FUNCTION_BLOCK FB_PackMLBase
VAR_INPUT
	PackMLIn	: ST_PML_Base_In;
	
	bEnable				: BOOL := TRUE;
	bExternalFault		: BOOL;
END_VAR
VAR_OUTPUT
	PackMLOut	: ST_PML_Base_Out;
	
	bTransitionActive	: BOOL;
END_VAR
VAR
	_eLastCommand			: E_PackMLCommand := E_PackMLCommand.None;
	_eCommandToProcess		: E_PackMLCommand := E_PackMLCommand.None;
	_eQueuedCommand			: E_PackMLCommand := E_PackMLCommand.None;
	_bQueuedCommandRequest	: BOOL;
	_bCommandConsumed		: BOOL;
	_bModeChangeConsumed	: BOOL;
	_bStateFirstScan		: BOOL := TRUE;
	_bStateFirstScanForHook	: BOOL;
	_eHookResult			: E_PackMLHookResult;
END_VAR

// Reset edge-style status before evaluating this PLC cycle.
_eCommandToProcess		:= E_PackMLCommand.None;

// Command and mode request feedback is latched for HMI/upper-layer handshakes
// until the corresponding request input returns to FALSE.
IF NOT PackMLIn.bCommandChangeRequest THEN
	PackMLOut.bCommandAccepted	:= FALSE;
	PackMLOut.bCommandRejected	:= FALSE;
	PackMLOut.eStateErrorID			:= E_PackMLErrorID.NoError;
END_IF

IF NOT PackMLIn.bModeChangeRequest THEN
	PackMLOut.bModeChanged		:= FALSE;
	PackMLOut.bModeChangeRejected	:= FALSE;
	PackMLOut.eModeErrorID		:= E_PackMLErrorID.NoError;
END_IF

// A disabled base FB holds the current state and suppresses transition activity.
IF NOT bEnable THEN
	bTransitionActive := FALSE;
	RETURN;
END_IF

// Mode change requests are edge/latch based, matching command request behavior.
// The caller must clear stIn.bModeChangeRequest before the same request can run again.
IF NOT PackMLIn.bModeChangeRequest THEN
	_bModeChangeConsumed := FALSE;
END_IF

IF PackMLIn.bModeChangeRequest AND NOT _bModeChangeConsumed THEN
	_bModeChangeConsumed := TRUE;

	IF NOT H_IsModeSupported(PackMLIn.eMode) THEN
		M_RejectModeChange(E_PackMLErrorID.ModeNotSupported);
	ELSIF PackMLIn.eMode = PackMLOut.eModeCurrent THEN
		M_RejectModeChange(E_PackMLErrorID.ModeAlreadyActive);
	ELSIF NOT M_IsModeChangeAllowedByState() THEN
		M_RejectModeChange(E_PackMLErrorID.ModeChangeNotAllowedFromCurrentState);
	ELSIF NOT H_IsStateSupportedByMode(PackMLIn.eMode, PackMLOut.eStateCurrent) THEN
		M_RejectModeChange(E_PackMLErrorID.ModeDoesNotSupportCurrentState);
	ELSE
		M_ChangeMode(PackMLIn.eMode);
	END_IF
END_IF

// Command requests are edge/latch based, matching mode-change request behavior.
// The caller must clear stIn.bCommandChangeRequest before another command can run.
IF NOT PackMLIn.bCommandChangeRequest THEN
	_bCommandConsumed	:= FALSE;
	_eLastCommand		:= E_PackMLCommand.None;
END_IF

// External faults have priority over normal commands and force the abort path
// only while the machine is not already Aborting or Aborted.
IF bExternalFault AND M_IsAbortAllowedByState() THEN
	_eCommandToProcess := E_PackMLCommand.Abort;
ELSIF _bQueuedCommandRequest AND (_eQueuedCommand <> E_PackMLCommand.None) THEN
	_eCommandToProcess		:= _eQueuedCommand;
	_eQueuedCommand			:= E_PackMLCommand.None;
	_bQueuedCommandRequest	:= FALSE;
ELSIF PackMLIn.bCommandChangeRequest AND (PackMLIn.eCommand <> E_PackMLCommand.None) AND NOT _bCommandConsumed THEN
	_eCommandToProcess	:= PackMLIn.eCommand;
	_eLastCommand		:= PackMLIn.eCommand;
	_bCommandConsumed	:= TRUE;
END_IF

// Mode policy hooks run before PackML state guards so a forbidden command reports
// the mode reason instead of a state reason.
IF (_eCommandToProcess <> E_PackMLCommand.None) AND NOT H_IsCommandAllowedByMode(_eCommandToProcess, PackMLOut.eModeCurrent) THEN
	M_RejectCommand(E_PackMLErrorID.CommandNotAllowedInActiveMode);
	_eCommandToProcess := E_PackMLCommand.None;
END_IF

// Dispatch the accepted command through private PackML state guards.
// Rejected commands never mutate the state and return a stable numeric error ID.
CASE _eCommandToProcess OF
	E_PackMLCommand.Clear:
		IF M_IsClearAllowedByState() THEN
			PackMLOut.bCommandAccepted := TRUE;
			M_ChangeState(E_PackMLState.Clearing);
		ELSE
			M_RejectCommand(E_PackMLErrorID.ClearNotAllowedFromCurrentState);
		END_IF

	E_PackMLCommand.Reset:
		IF M_IsResetAllowedByState() THEN
			PackMLOut.bCommandAccepted := TRUE;
			M_ChangeState(E_PackMLState.Resetting);
		ELSE
			M_RejectCommand(E_PackMLErrorID.ResetNotAllowedFromCurrentState);
		END_IF

	E_PackMLCommand.Start:
		IF M_IsStartAllowedByState() THEN
			PackMLOut.bCommandAccepted := TRUE;
			M_ChangeState(E_PackMLState.Starting);
		ELSE
			M_RejectCommand(E_PackMLErrorID.StartNotAllowedFromCurrentState);
		END_IF

	E_PackMLCommand.Stop:
		IF M_IsStopAllowedByState() THEN
			PackMLOut.bCommandAccepted := TRUE;
			M_ChangeState(E_PackMLState.Stopping);
		ELSE
			M_RejectCommand(E_PackMLErrorID.StopNotAllowedFromCurrentState);
		END_IF

	E_PackMLCommand.Hold:
		IF M_IsHoldAllowedByState() THEN
			PackMLOut.bCommandAccepted := TRUE;
			M_ChangeState(E_PackMLState.Holding);
		ELSE
			M_RejectCommand(E_PackMLErrorID.HoldNotAllowedFromCurrentState);
		END_IF

	E_PackMLCommand.Unhold:
		IF M_IsUnholdAllowedByState() THEN
			PackMLOut.bCommandAccepted := TRUE;
			M_ChangeState(E_PackMLState.Unholding);
		ELSE
			M_RejectCommand(E_PackMLErrorID.UnholdNotAllowedFromCurrentState);
		END_IF

	E_PackMLCommand.Suspend:
		IF M_IsSuspendAllowedByState() THEN
			PackMLOut.bCommandAccepted := TRUE;
			M_ChangeState(E_PackMLState.Suspending);
		ELSE
			M_RejectCommand(E_PackMLErrorID.SuspendNotAllowedFromCurrentState);
		END_IF

	E_PackMLCommand.Unsuspend:
		IF M_IsUnsuspendAllowedByState() THEN
			PackMLOut.bCommandAccepted := TRUE;
			M_ChangeState(E_PackMLState.Unsuspending);
		ELSE
			M_RejectCommand(E_PackMLErrorID.UnsuspendNotAllowedFromCurrentState);
		END_IF

	E_PackMLCommand.Abort:
		IF M_IsAbortAllowedByState() THEN
			PackMLOut.bCommandAccepted := TRUE;
			M_ChangeState(E_PackMLState.Aborting);
		ELSE
			M_RejectCommand(E_PackMLErrorID.AbortNotAllowedFromCurrentState);
		END_IF
END_CASE

// Run the current state's action hook, then advance transient states when their
// hook reports Done. Stable states remain active until a command moves them.
_bStateFirstScanForHook	:= _bStateFirstScan;
_bStateFirstScan		:= FALSE;

CASE PackMLOut.eStateCurrent OF
	E_PackMLState.Undefined:
		_eHookResult := H_OnUndefined(_bStateFirstScanForHook);
		IF _eHookResult = E_PackMLHookResult.Done THEN
			M_ChangeState(E_PackMLState.Aborted);
		END_IF

	E_PackMLState.Clearing:
		_eHookResult := H_OnClearing(_bStateFirstScanForHook);
		IF _eHookResult = E_PackMLHookResult.Done THEN
			M_ChangeState(E_PackMLState.Stopped);
		END_IF

	E_PackMLState.Stopped:
		H_OnStopped(_bStateFirstScanForHook);

	E_PackMLState.Starting:
		_eHookResult := H_OnStarting(_bStateFirstScanForHook);
		IF _eHookResult = E_PackMLHookResult.Done THEN
			M_ChangeState(E_PackMLState.Execute);
		END_IF

	E_PackMLState.Idle:
		H_OnIdle(_bStateFirstScanForHook);

	E_PackMLState.Suspended:
		H_OnSuspended(_bStateFirstScanForHook);

	E_PackMLState.Execute:
		_eHookResult := H_OnExecute(_bStateFirstScanForHook);
		IF _eHookResult = E_PackMLHookResult.Done THEN
			M_ChangeState(E_PackMLState.Completing);
		END_IF

	E_PackMLState.Stopping:
		_eHookResult := H_OnStopping(_bStateFirstScanForHook);
		IF _eHookResult = E_PackMLHookResult.Done THEN
			M_ChangeState(E_PackMLState.Stopped);
		END_IF

	E_PackMLState.Aborting:
		_eHookResult := H_OnAborting(_bStateFirstScanForHook);
		IF _eHookResult = E_PackMLHookResult.Done THEN
			M_ChangeState(E_PackMLState.Aborted);
		END_IF

	E_PackMLState.Aborted:
		H_OnAborted(_bStateFirstScanForHook);

	E_PackMLState.Holding:
		_eHookResult := H_OnHolding(_bStateFirstScanForHook);
		IF _eHookResult = E_PackMLHookResult.Done THEN
			M_ChangeState(E_PackMLState.Held);
		END_IF

	E_PackMLState.Held:
		H_OnHeld(_bStateFirstScanForHook);

	E_PackMLState.Unholding:
		_eHookResult := H_OnUnholding(_bStateFirstScanForHook);
		IF _eHookResult = E_PackMLHookResult.Done THEN
			M_ChangeState(E_PackMLState.Execute);
		END_IF

	E_PackMLState.Suspending:
		_eHookResult := H_OnSuspending(_bStateFirstScanForHook);
		IF _eHookResult = E_PackMLHookResult.Done THEN
			M_ChangeState(E_PackMLState.Suspended);
		END_IF

	E_PackMLState.Unsuspending:
		_eHookResult := H_OnUnsuspending(_bStateFirstScanForHook);
		IF _eHookResult = E_PackMLHookResult.Done THEN
			M_ChangeState(E_PackMLState.Execute);
		END_IF

	E_PackMLState.Resetting:
		_eHookResult := H_OnResetting(_bStateFirstScanForHook);
		IF _eHookResult = E_PackMLHookResult.Done THEN
			M_ChangeState(E_PackMLState.Idle);
		END_IF

	E_PackMLState.Completing:
		_eHookResult := H_OnCompleting(_bStateFirstScanForHook);
		IF _eHookResult = E_PackMLHookResult.Done THEN
			M_ChangeState(E_PackMLState.Complete);
		END_IF

	E_PackMLState.Complete:
		H_OnComplete(_bStateFirstScanForHook);
END_CASE

// Transition activity is true for transient states that normally need completion
// confirmation from their state hook.
bTransitionActive :=
	(PackMLOut.eStateCurrent = E_PackMLState.Undefined) OR
	(PackMLOut.eStateCurrent = E_PackMLState.Clearing) OR
	(PackMLOut.eStateCurrent = E_PackMLState.Starting) OR
	(PackMLOut.eStateCurrent = E_PackMLState.Stopping) OR
	(PackMLOut.eStateCurrent = E_PackMLState.Aborting) OR
	(PackMLOut.eStateCurrent = E_PackMLState.Holding) OR
	(PackMLOut.eStateCurrent = E_PackMLState.Unholding) OR
	(PackMLOut.eStateCurrent = E_PackMLState.Suspending) OR
	(PackMLOut.eStateCurrent = E_PackMLState.Unsuspending) OR
	(PackMLOut.eStateCurrent = E_PackMLState.Resetting) OR
	(PackMLOut.eStateCurrent = E_PackMLState.Completing);

METHOD PROTECTED H_IsCommandAllowedByMode : BOOL
VAR_INPUT
	eRequestedCommand	: E_PackMLCommand;
	eActiveMode			: T_PackMLMode;
END_VAR
// Modes are application-defined in library use; override to restrict commands per mode.
H_IsCommandAllowedByMode := TRUE;
END_METHOD

METHOD PROTECTED H_IsModeSupported : BOOL
VAR_INPUT
	eRequestedMode	: T_PackMLMode;
END_VAR
// Modes are application-defined in library use; override to reject unsupported modes.
H_IsModeSupported := TRUE;
END_METHOD

METHOD PROTECTED H_IsStateSupportedByMode : BOOL
VAR_INPUT
	eRequestedMode	: T_PackMLMode;
	eCurrentState	: E_PackMLState;
END_VAR
// Modes are application-defined in library use; override to restrict mode/state pairs.
H_IsStateSupportedByMode := TRUE;
END_METHOD

METHOD PROTECTED H_OnAborted
VAR_INPUT
	bFirstScan	: BOOL;
END_VAR
// Default action hook intentionally empty. Override in derived FBs when needed.
END_METHOD

METHOD PROTECTED H_OnAborting : E_PackMLHookResult
VAR_INPUT
	bFirstScan	: BOOL;
END_VAR
// Default transient hooks complete immediately; override when work is required.
H_OnAborting := E_PackMLHookResult.Done;
END_METHOD

METHOD PROTECTED H_OnClearing : E_PackMLHookResult
VAR_INPUT
	bFirstScan	: BOOL;
END_VAR
// Default transient hooks complete immediately; override when work is required.
H_OnClearing := E_PackMLHookResult.Done;
END_METHOD

METHOD PROTECTED H_OnComplete
VAR_INPUT
	bFirstScan	: BOOL;
END_VAR
// Default action hook intentionally empty. Override in derived FBs when needed.
END_METHOD

METHOD PROTECTED H_OnCompleting : E_PackMLHookResult
VAR_INPUT
	bFirstScan	: BOOL;
END_VAR
// Default transient hooks complete immediately; override when work is required.
H_OnCompleting := E_PackMLHookResult.Done;
END_METHOD

METHOD PROTECTED H_OnExecute : E_PackMLHookResult
VAR_INPUT
	bFirstScan	: BOOL;
END_VAR
// Execute is stable by default; derived FBs decide when the process is done.
H_OnExecute := E_PackMLHookResult.Busy;
END_METHOD

METHOD PROTECTED H_OnHeld
VAR_INPUT
	bFirstScan	: BOOL;
END_VAR
// Default action hook intentionally empty. Override in derived FBs when needed.
END_METHOD

METHOD PROTECTED H_OnHolding : E_PackMLHookResult
VAR_INPUT
	bFirstScan	: BOOL;
END_VAR
// Default transient hooks complete immediately; override when work is required.
H_OnHolding := E_PackMLHookResult.Done;
END_METHOD

METHOD PROTECTED H_OnIdle
VAR_INPUT
	bFirstScan	: BOOL;
END_VAR
// Default action hook intentionally empty. Override in derived FBs when needed.
END_METHOD

METHOD PROTECTED H_OnModeChanged
VAR_INPUT
	ePreviousMode	: T_PackMLMode;
	eNewMode		: T_PackMLMode;
END_VAR
// Default mode-change hook intentionally empty. Override in derived FBs when needed.
END_METHOD

METHOD PROTECTED H_OnResetting : E_PackMLHookResult
VAR_INPUT
	bFirstScan	: BOOL;
END_VAR
// Default transient hooks complete immediately; override when work is required.
H_OnResetting := E_PackMLHookResult.Done;
END_METHOD

METHOD PROTECTED H_OnStarting : E_PackMLHookResult
VAR_INPUT
	bFirstScan	: BOOL;
END_VAR
// Default transient hooks complete immediately; override when work is required.
H_OnStarting := E_PackMLHookResult.Done;
END_METHOD

METHOD PROTECTED H_OnStateChanged
VAR_INPUT
	ePreviousState	: E_PackMLState;
	eNewState		: E_PackMLState;
END_VAR
// Default state-change hook intentionally empty. Override in derived FBs when needed.
END_METHOD

METHOD PROTECTED H_OnStopped
VAR_INPUT
	bFirstScan	: BOOL;
END_VAR
// Default action hook intentionally empty. Override in derived FBs when needed.
END_METHOD

METHOD PROTECTED H_OnStopping : E_PackMLHookResult
VAR_INPUT
	bFirstScan	: BOOL;
END_VAR
// Default transient hooks complete immediately; override when work is required.
H_OnStopping := E_PackMLHookResult.Done;
END_METHOD

METHOD PROTECTED H_OnSuspended
VAR_INPUT
	bFirstScan	: BOOL;
END_VAR
// Default action hook intentionally empty. Override in derived FBs when needed.
END_METHOD

METHOD PROTECTED H_OnSuspending : E_PackMLHookResult
VAR_INPUT
	bFirstScan	: BOOL;
END_VAR
// Default transient hooks complete immediately; override when work is required.
H_OnSuspending := E_PackMLHookResult.Done;
END_METHOD

METHOD PROTECTED H_OnUndefined : E_PackMLHookResult
VAR_INPUT
	bFirstScan	: BOOL;
END_VAR
// The base FB leaves Undefined immediately unless a derived FB delays startup.
H_OnUndefined := E_PackMLHookResult.Done;
END_METHOD

METHOD PROTECTED H_OnUnholding : E_PackMLHookResult
VAR_INPUT
	bFirstScan	: BOOL;
END_VAR
// Default transient hooks complete immediately; override when work is required.
H_OnUnholding := E_PackMLHookResult.Done;
END_METHOD

METHOD PROTECTED H_OnUnsuspending : E_PackMLHookResult
VAR_INPUT
	bFirstScan	: BOOL;
END_VAR
// Default transient hooks complete immediately; override when work is required.
H_OnUnsuspending := E_PackMLHookResult.Done;
END_METHOD

METHOD PRIVATE M_ChangeMode
VAR_INPUT
	eNextMode	: T_PackMLMode;
END_VAR
// Centralize mode mutation so previous-mode and edge outputs stay consistent.
IF PackMLOut.eModeCurrent <> eNextMode THEN
	PackMLOut.eModePrevious	:= PackMLOut.eModeCurrent;
	PackMLOut.eModeCurrent	:= eNextMode;
	PackMLOut.bModeChanged	:= TRUE;
	H_OnModeChanged(PackMLOut.eModePrevious, PackMLOut.eModeCurrent);
END_IF
END_METHOD

METHOD PRIVATE M_ChangeState
VAR_INPUT
	eNextState	: E_PackMLState;
END_VAR
// Centralize state mutation so previous-state and edge outputs stay consistent.
IF PackMLOut.eStateCurrent <> eNextState THEN
	PackMLOut.eStatePrevious	:= PackMLOut.eStateCurrent;
	PackMLOut.eStateCurrent			:= eNextState;
	_bStateFirstScan			:= TRUE;
	H_OnStateChanged(PackMLOut.eStatePrevious, PackMLOut.eStateCurrent);
END_IF
END_METHOD

METHOD PRIVATE M_IsAbortAllowedByState : BOOL
// Abort is valid from every state except the terminal abort states.
M_IsAbortAllowedByState := (PackMLOut.eStateCurrent <> E_PackMLState.Aborting) AND (PackMLOut.eStateCurrent <> E_PackMLState.Aborted);
END_METHOD

METHOD PRIVATE M_IsClearAllowedByState : BOOL
// Clear leaves the safe Aborted state and starts the resettable stop path.
M_IsClearAllowedByState := PackMLOut.eStateCurrent = E_PackMLState.Aborted;
END_METHOD

METHOD PRIVATE M_IsCompleteAllowedByState : BOOL
// Complete is only meaningful while the unit is executing.
M_IsCompleteAllowedByState := PackMLOut.eStateCurrent = E_PackMLState.Execute;
END_METHOD

METHOD PRIVATE M_IsHoldAllowedByState : BOOL
// Hold pauses an active Execute flow.
M_IsHoldAllowedByState := PackMLOut.eStateCurrent = E_PackMLState.Execute;
END_METHOD

METHOD PRIVATE M_IsModeChangeAllowedByState : BOOL
// Mode changes can only be attempted from safe stable states.
// Target mode compatibility is checked separately after this safety gate.
// Henry: Bypass "Held" & "Suspended" state due to consideration about state-related parameters inconsistent
M_IsModeChangeAllowedByState :=
	(PackMLOut.eStateCurrent = E_PackMLState.Aborted) OR
	(PackMLOut.eStateCurrent = E_PackMLState.Stopped) OR
	(PackMLOut.eStateCurrent = E_PackMLState.Idle) OR
	(PackMLOut.eStateCurrent = E_PackMLState.Complete);
END_METHOD

METHOD PRIVATE M_IsResetAllowedByState : BOOL
// Reset prepares the unit from Stopped or Complete into Idle.
M_IsResetAllowedByState := (PackMLOut.eStateCurrent = E_PackMLState.Stopped) OR (PackMLOut.eStateCurrent = E_PackMLState.Complete);
END_METHOD

METHOD PRIVATE M_IsStartAllowedByState : BOOL
// Start begins production or operation only from Idle.
M_IsStartAllowedByState := PackMLOut.eStateCurrent = E_PackMLState.Idle;
END_METHOD

METHOD PRIVATE M_IsStopAllowedByState : BOOL
// Stop is accepted from normal operating, paused, and completing states.
M_IsStopAllowedByState :=
	(PackMLOut.eStateCurrent = E_PackMLState.Starting) OR
	(PackMLOut.eStateCurrent = E_PackMLState.Idle) OR
	(PackMLOut.eStateCurrent = E_PackMLState.Execute) OR
	(PackMLOut.eStateCurrent = E_PackMLState.Completing) OR
	(PackMLOut.eStateCurrent = E_PackMLState.Complete) OR
	(PackMLOut.eStateCurrent = E_PackMLState.Holding) OR
	(PackMLOut.eStateCurrent = E_PackMLState.Held) OR
	(PackMLOut.eStateCurrent = E_PackMLState.Unholding) OR
	(PackMLOut.eStateCurrent = E_PackMLState.Suspending) OR
	(PackMLOut.eStateCurrent = E_PackMLState.Suspended) OR
	(PackMLOut.eStateCurrent = E_PackMLState.Unsuspending);
END_METHOD

METHOD PRIVATE M_IsSuspendAllowedByState : BOOL
// Suspend pauses Execute because of an external process condition.
M_IsSuspendAllowedByState := PackMLOut.eStateCurrent = E_PackMLState.Execute;
END_METHOD

METHOD PRIVATE M_IsUnholdAllowedByState : BOOL
// Unhold resumes from the stable Held state.
M_IsUnholdAllowedByState := PackMLOut.eStateCurrent = E_PackMLState.Held;
END_METHOD

METHOD PRIVATE M_IsUnsuspendAllowedByState : BOOL
// Unsuspend resumes from the stable Suspended state.
M_IsUnsuspendAllowedByState := PackMLOut.eStateCurrent = E_PackMLState.Suspended;
END_METHOD

METHOD PRIVATE M_RejectCommand
VAR_INPUT
	eErrorID	: E_PackMLErrorID;
END_VAR
// Centralize rejected-command reporting so every guard failure has a stable ID.
PackMLOut.bCommandRejected	:= TRUE;
PackMLOut.eStateErrorID		:= eErrorID;
END_METHOD

METHOD PRIVATE M_RejectModeChange
VAR_INPUT
	eErrorID	: E_PackMLErrorID;
END_VAR
// Keep mode-change errors separate from PackML command/state errors.
PackMLOut.bModeChangeRejected	:= TRUE;
PackMLOut.eModeErrorID		:= eErrorID;
END_METHOD

// Used for requesting PackML command inside state machine itself 
METHOD PROTECTED RequestCommand : BOOL
VAR_INPUT
	eTargetCmd	: E_PackMLCommand;
END_VAR
RequestCommand := FALSE;

IF _bQueuedCommandRequest OR PackMLIn.bModeChangeRequest THEN
	RETURN;
END_IF

_eQueuedCommand			:= eTargetCmd;
_bQueuedCommandRequest	:= TRUE;
RequestCommand := TRUE;
END_METHOD

END_FUNCTION_BLOCK

(* stored: Version 1.1.0.1, ProductVersion 3.1.4026.18
   POU FB_PackMLBase: Id {bb7074bb-cd46-4555-9ada-1eb1c7832876}, SpecialFunc None
   Folder Mode Setting Hook Method: Id {804b7073-8ed6-4fb6-a676-84629a6495bf}
   Folder Private Method: Id {82a24892-a715-46be-9ec0-bcb60939def2}
   Folder State Action Hook Method: Id {d761a877-4908-4619-b1fa-1df698a584cd}
   Folder Useful Hook Method: Id {3cc24201-1b27-4b01-89a9-bc66f9f103ef}
   Method H_IsCommandAllowedByMode: Id {9a833552-ec23-421d-885d-93766f9e9ef6}
   Method H_IsModeSupported: Id {5a131af6-fe63-4452-b7b9-fbb87cf32720}
   Method H_IsStateSupportedByMode: Id {8ecb8812-d961-4d2e-a8cf-d988ced19232}
   Method H_OnAborted: Id {4bb17b66-fb2e-4627-9258-890a485508f8}
   Method H_OnAborting: Id {a13be449-422e-4d8b-8327-e77d3d480251}
   Method H_OnClearing: Id {3403ef10-749e-425d-81c7-aa09980fc7da}
   Method H_OnComplete: Id {c6c044b2-0836-4192-a54d-4875856d12b0}
   Method H_OnCompleting: Id {b3c87bff-3a95-4825-9f3e-aed9464089fa}
   Method H_OnExecute: Id {b44dc1df-23a6-4acf-aaac-94c4f43cef35}
   Method H_OnHeld: Id {44f5e96b-d14a-41e4-981a-73134384adb2}
   Method H_OnHolding: Id {3c2f9be6-b71e-4397-8e36-22ce7a5cf40a}
   Method H_OnIdle: Id {e8d1bb5c-d66f-4b90-80aa-5521f4b1e39c}
   Method H_OnModeChanged: Id {5e0980df-e69c-424a-be57-a8bf711b5d04}
   Method H_OnResetting: Id {19822229-7b7e-42d6-b9ad-fdcdb660e283}
   Method H_OnStarting: Id {d244760c-0e73-42e0-9524-ef70583c8446}
   Method H_OnStateChanged: Id {b39fd166-f67a-4543-bd9f-b74320073c49}
   Method H_OnStopped: Id {95c75646-2932-442e-99c7-630b54b18d98}
   Method H_OnStopping: Id {b44aa23e-e863-41e5-8d65-5b23b51b1809}
   Method H_OnSuspended: Id {af02e98b-4ca8-4346-9586-599f47a3f0c8}
   Method H_OnSuspending: Id {7a0bfcb6-56b3-492b-86a5-8cc3ec32e492}
   Method H_OnUndefined: Id {348c6696-4691-4303-b7e8-15f37a1c30ff}
   Method H_OnUnholding: Id {900cc882-799f-423d-876a-12412604b19e}
   Method H_OnUnsuspending: Id {d4125dcf-e5e7-4271-a103-073060450909}
   Method M_ChangeMode: Id {480596f8-48a1-425b-a307-21512e84f091}
   Method M_ChangeState: Id {bf78a96d-9d4e-42b6-b159-e367e8ad7c2c}
   Method M_IsAbortAllowedByState: Id {fa7a4de6-c9e7-4315-9d09-7067965a2941}
   Method M_IsClearAllowedByState: Id {332a91a0-3733-42b2-abec-4c14a54021cd}
   Method M_IsCompleteAllowedByState: Id {e29a4438-6687-4116-a4d4-577056243d8b}
   Method M_IsHoldAllowedByState: Id {49bde5a5-35d4-4747-a469-fc23b21ffacd}
   Method M_IsModeChangeAllowedByState: Id {5a21c016-dfdc-4c29-86e7-52905f19cfbd}
   Method M_IsResetAllowedByState: Id {38b5684f-4df4-4061-acdd-f532c5411342}
   Method M_IsStartAllowedByState: Id {5a2e9cc0-9e0d-4da4-a55b-a165f1eeb9bf}
   Method M_IsStopAllowedByState: Id {f0da80f2-c0a2-4ca1-a63e-a5b90bf2f04c}
   Method M_IsSuspendAllowedByState: Id {362e955c-d91e-4573-ac49-5e1f5561e9d1}
   Method M_IsUnholdAllowedByState: Id {90276ba7-ddef-4e56-8b6f-9f76fe99435a}
   Method M_IsUnsuspendAllowedByState: Id {c3563b72-aa8b-4b4c-9d01-38e261429a17}
   Method M_RejectCommand: Id {fd9fdbf3-d906-4767-8436-2bb609e1c84f}
   Method M_RejectModeChange: Id {424b9d75-e7ad-40d7-b41a-b08d033526d2}
   Method RequestCommand: Id {acc2f90f-ee3a-48ba-968f-939630ff093a} *)
